(* PLC project  *)

CONFIGURATION Robot_C
END_CONFIGURATION
